Staubli VAL3: cycle_version.pgx

program cycle_version()
  local num i
  local num j
  local num l_hours
  local string l_sMessage
begin
  //
  // template Version status
  //
  if getVersion("valTending")!="enabled"
    //
    l_hours=roundDown(clock()/3600000)
    if l_hours>=2
      cycleStatus:nToSuperV=4
      call language:message(l_sMessage,230)
      popUpMsg(l_sMessage)
      cycleStatus:bToStop=true
    endIf
  endIf
end
